// TIA Portal project "FactoryIO_scene3_fillingTank" (V16)

(* hardware
DEVICE "S7-1200 station_1"  S7-1200 Station
   slot 0: "Rack_0"  S7-1200 Rack  Rack  V1.0
   slot 1: "PLC_1"  CPU 1214C DC/DC/DC  6ES7 214-1AG40-0XB0  V4.4
*)

// ===== PLC "PLC_1"  CPU 1214C DC/DC/DC =====

VAR_GLOBAL   // PLC tag table "Default tag table"
   "Tag_1" AT %M0.0 : Bool;
   "Tag_2" AT %M0.1 : Bool;
   "Tag_3" AT %M0.2 : Bool;
END_VAR

VAR_GLOBAL   // PLC tag table "IO_tags"
   "fill" AT %I0.0 : Bool;
   "Discharge" AT %I0.1 : Bool;
   "Factory IO running" AT %I0.2 : Bool;
   "filll valve" AT %Q0.0 : Bool;
   "filling" AT %Q0.1 : Bool;
   "discharge valve" AT %Q0.2 : Bool;
   "discharging" AT %Q0.3 : Bool;
   "Timer" AT %QD30 : DInt;
END_VAR

DATA_BLOCK "data"   // DB4
{ S7_Optimized_Access := 'TRUE' }
VERSION : 0.1
   VAR
      fill_time : Time;
      discharge_time : Time;
   END_VAR
BEGIN
END_DATA_BLOCK

// folder: System blocks/Program resources

DATA_BLOCK "Discharge Timer"   // DB1
{ S7_Optimized_Access := 'TRUE' }
AUTHOR : Simatic
FAMILY : IEC
NAME : IEC_TMR
VERSION : 1.0
// stored: InstanceOfName IEC_TIMER
"IEC_TIMER"
BEGIN
END_DATA_BLOCK

DATA_BLOCK "fill timer"   // DB5
{ S7_Optimized_Access := 'TRUE' }
AUTHOR : Simatic
FAMILY : IEC
NAME : IEC_TMR
VERSION : 1.0
// stored: InstanceOfName IEC_TIMER
"IEC_TIMER"
BEGIN
END_DATA_BLOCK

// folder: (top level)

FUNCTION "MHJ-PLC-Lab-Function-S71200" : Void   // FC9000, SCL
{ S7_Optimized_Access := 'TRUE' }
VERSION : 0.1
   VAR_TEMP
      rdTimeReturn : Int;
      outputTime : DTL;
      SyncVal : Byte;
      forVal : Int;
      forVal_2 : Int;
      Value : Byte;
   END_VAR
   VAR CONSTANT
      CompVal : Byte := 16#34;
      Value_01 : Byte := 16#11;
      Value_01_DW : DWord := 16#A165_D992;
      Value_02_DW : DWord := 16#58BE_4401;
   END_VAR
BEGIN

   #Value:=PEEK(area := 16#82,
        dbNumber := 0,
        byteOffset := 511);
   #Value := #Value + 1;

   POKE(area := 16#82,
        dbNumber := 0,
        byteOffset := 511,
        value := #Value);

   POKE(area:=16#81,
        dbNumber:=0,
        byteOffset:=1016,
        value:=#Value_01_DW);
   POKE(area := 16#81,
        dbNumber := 0,
        byteOffset := 1020,
        value := #Value_02_DW);

   POKE(area := 16#81,
        dbNumber := 0,
        byteOffset := 511,
        value := B#16#00);

   FOR #forVal := 0 TO 120 DO
       FOR #forVal_2:=0 TO 10 DO
           #rdTimeReturn:=RD_SYS_T(#outputTime);
           #rdTimeReturn := WR_SYS_T(#outputTime);
           #rdTimeReturn := RD_SYS_T(#outputTime);
           #rdTimeReturn := WR_SYS_T(#outputTime);
       END_FOR;
       #SyncVal:= PEEK(area := 16#81,
                      dbNumber := 0,
                      byteOffset := 511);
       IF #SyncVal = #CompVal THEN
          GOTO M_1;
       END_IF;
   END_FOR;
   RETURN;

   M_1:
   POKE(area := 16#81,
        dbNumber := 0,
        byteOffset := 511,
        value := B#16#0);
END_FUNCTION

ORGANIZATION_BLOCK "Main"   // OB1, LAD, ProgramCycle
TITLE = "Main Program Sweep (Cycle)"
{ S7_Optimized_Access := 'TRUE' }
VERSION : 0.1
   VAR_INPUT
      Initial_Call : Bool;   // Initial call of this OB
      Remanence : Bool;   // =True, if remanent data are available
   END_VAR
   VAR_TEMP
      current_step : Int;
      reset : Bool;
   END_VAR
   VAR CONSTANT
      box_count : Int := 3;   // Number of buffer boxes
   END_VAR
BEGIN

REGION Network 1
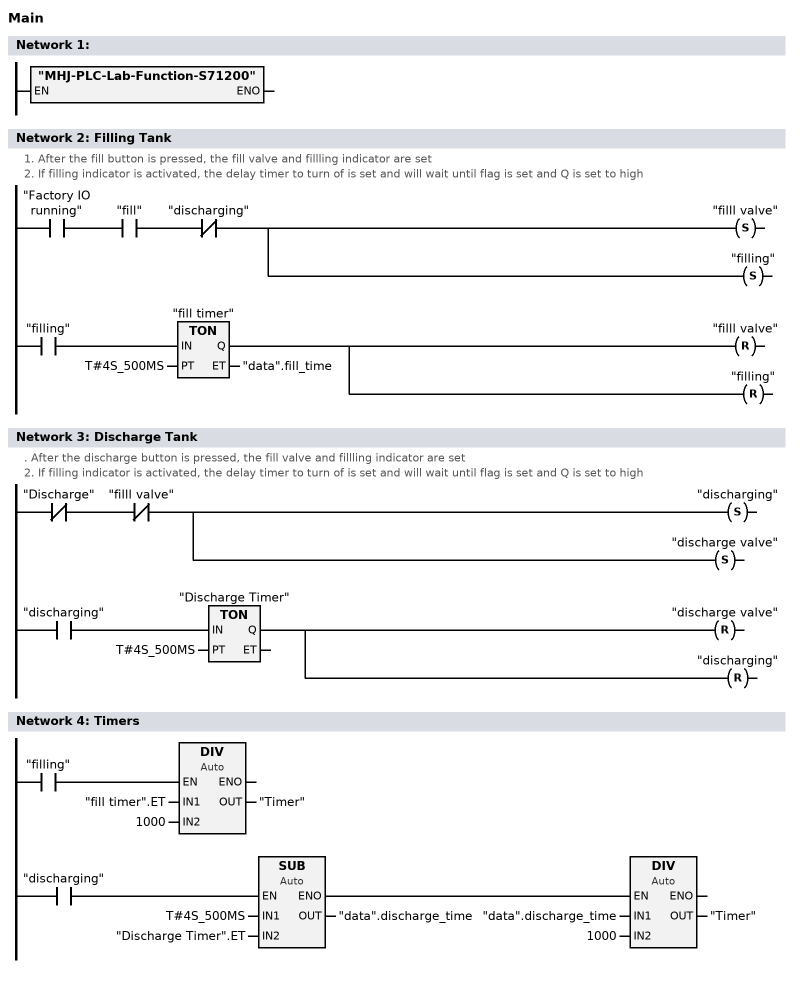
   RUNG wire#powerrail
      "MHJ-PLC-Lab-Function-S71200"()
   END_RUNG
   // the same network as SCL:
   "MHJ-PLC-Lab-Function-S71200"();
END_REGION

REGION Network 2: Filling Tank
   // 1. After the fill button is pressed, the fill valve and fillling indicator are set
   // 2. If filling indicator is activated, the delay timer to turn of is set and will wait until flag is set and Q is set to high
   IF "Factory IO running" AND "fill" AND NOT "discharging" THEN
       "filll valve" := TRUE;
       "filling" := TRUE;
   END_IF;
   "fill timer".TON(IN := "filling", PT := T#4S_500MS, ET => "data".fill_time);
   IF "fill timer".Q THEN
       "filll valve" := FALSE;
       "filling" := FALSE;
   END_IF;
END_REGION

REGION Network 3: Discharge Tank
   // . After the discharge button is pressed, the fill valve and fillling indicator are set
   // 2. If filling indicator is activated, the delay timer to turn of is set and will wait until flag is set and Q is set to high
   IF NOT "Discharge" AND NOT "filll valve" THEN
       "discharging" := TRUE;
       "discharge valve" := TRUE;
   END_IF;
   "Discharge Timer".TON(IN := "discharging", PT := T#4S_500MS);
   IF "Discharge Timer".Q THEN
       "discharge valve" := FALSE;
       "discharging" := FALSE;
   END_IF;
END_REGION

REGION Network 4: Timers
   RUNG wire#powerrail
      Contact( "filling" )
      Div(in1 := "fill timer".ET, in2 := 1000, out => "Timer")
   END_RUNG
   RUNG wire#powerrail
      Contact( "discharging" )
      Sub(in1 := T#4S_500MS, in2 := "Discharge Timer".ET, out => "data".discharge_time)
      Div(in1 := "data".discharge_time, in2 := 1000, out => "Timer")
   END_RUNG
   // the same network as SCL:
   IF "filling" THEN "Timer" := "fill timer".ET / 1000; END_IF;
   IF "discharging" THEN
       "data".discharge_time := T#4S_500MS - "Discharge Timer".ET;
       "Timer" := "data".discharge_time / 1000;
   END_IF;
END_REGION
END_ORGANIZATION_BLOCK